INTERFACE ITest

METHOD Execute : BOOL
VAR_INPUT
END_VAR
END_METHOD

METHOD FB_init : BOOL
VAR_INPUT
	bInitRetains : BOOL; // if TRUE, the retain variables are initialized (warm start / cold start)
	bInCopyCode : BOOL;  // if TRUE, the instance afterwards gets moved into the copy code (online change)
	sName : STRING;
END_VAR
END_METHOD

PROPERTY Message : STRING[255]
GET
END_GET
END_PROPERTY

PROPERTY Name : STRING
GET
END_GET
END_PROPERTY

END_INTERFACE

(* stored: Version 1.1.0.1, ProductVersion 3.1.4024.12
   Itf ITest: Id {863de611-8c69-429c-b9f7-38b8134fde48}
   Method Execute: Id {0b8eec86-751b-4170-a607-88531178fdee}
   Method FB_init: Id {ceb96994-f34a-4fa5-9dc7-819eaab091ef}
   Property Message: Id {43ebdb2b-73be-4b99-a1ef-e5239f7d2566}
   Get Get: Id {ad9611f4-0769-47ff-8696-79774f3ed686}
   Property Name: Id {76ff6cfc-a6f9-4226-9f40-d82e74075ea0}
   Get Get: Id {35ae43ed-a6d7-4832-a9c5-86c369a5d73f} *)
